(* Schneider Machine Expert - Basic project memory words, file version 2.0.0.0 *)
(* ProjectInformations: Name=New project *)

HARDWARE
  Cpu 0: TM221CE16R
  EthernetConfiguration: NetworkName=M221, IpAllocationMode=FixedAddress, IpAddress=0.0.0.0, SubnetMask=0.0.0.0
  SerialLineConfiguration: Baud=Baud19200, Parity=ParityEven, DataBits=DataBits8, StopBits=StopBits1, PhysicalMedium=PhysicalMediumRs485, TransmissionMode=TransmissionModeModbusRtu, SlaveId=1, Addressing=SlaveAddressing
  MastTask: UsePeriodScanMode=false, PeriodScan=100
  FastTask: Period=255
  CpuBehavior: StartingMode=StartAsPreviousState, AutoSaveRamOnEeprom=true, WatchdogPeriod=250

SYMBOLS  (address, symbol, comment, settings)

POU New POU
  (* SectionNumber=1 *)

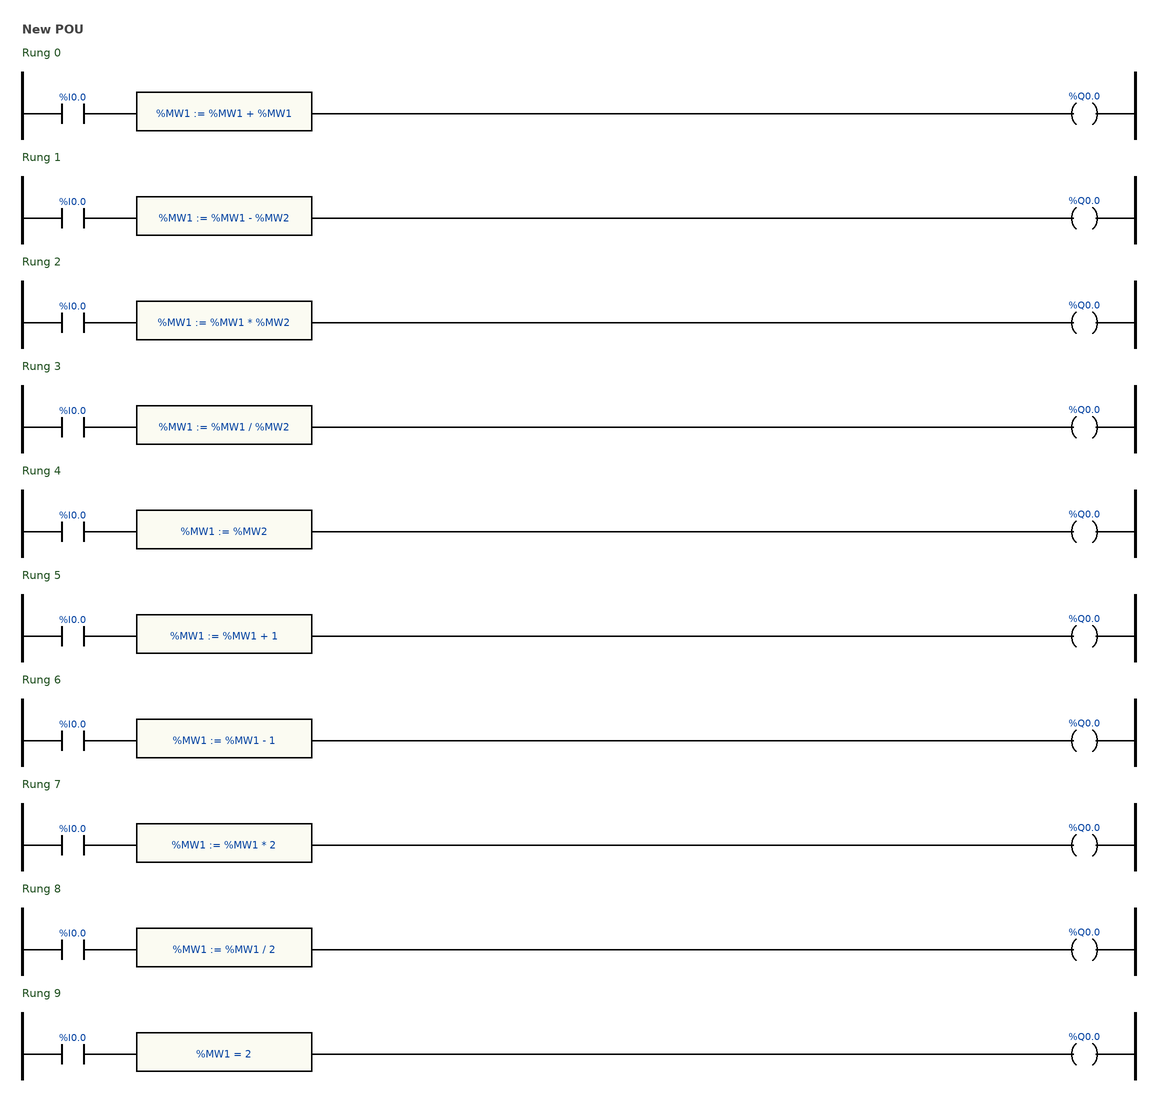

// Rung 0
  LD %I0.0
  OPER [ %MW1 := %MW1 + %MW1 ]
  ST %Q0.0
  // as ST:
  //   IF %I0.0 THEN %MW1 := %MW1 + %MW1; END_IF;
  //   %Q0.0 := %I0.0;

// Rung 1
  LD %I0.0
  OPER [ %MW1 := %MW1 - %MW2 ]
  ST %Q0.0
  // as ST:
  //   IF %I0.0 THEN %MW1 := %MW1 - %MW2; END_IF;
  //   %Q0.0 := %I0.0;

// Rung 2
  LD %I0.0
  OPER [ %MW1 := %MW1 * %MW2 ]
  ST %Q0.0
  // as ST:
  //   IF %I0.0 THEN %MW1 := %MW1 * %MW2; END_IF;
  //   %Q0.0 := %I0.0;

// Rung 3
  LD %I0.0
  OPER [ %MW1 := %MW1 / %MW2 ]
  ST %Q0.0
  // as ST:
  //   IF %I0.0 THEN %MW1 := %MW1 / %MW2; END_IF;
  //   %Q0.0 := %I0.0;

// Rung 4
  LD %I0.0
  OPER [ %MW1 := %MW2 ]
  ST %Q0.0
  // as ST:
  //   IF %I0.0 THEN %MW1 := %MW2; END_IF;
  //   %Q0.0 := %I0.0;

// Rung 5
  LD %I0.0
  OPER [ %MW1 := %MW1 + 1 ]
  ST %Q0.0
  // as ST:
  //   IF %I0.0 THEN %MW1 := %MW1 + 1; END_IF;
  //   %Q0.0 := %I0.0;

// Rung 6
  LD %I0.0
  OPER [ %MW1 := %MW1 - 1 ]
  ST %Q0.0
  // as ST:
  //   IF %I0.0 THEN %MW1 := %MW1 - 1; END_IF;
  //   %Q0.0 := %I0.0;

// Rung 7
  LD %I0.0
  OPER [ %MW1 := %MW1 * 2 ]
  ST %Q0.0
  // as ST:
  //   IF %I0.0 THEN %MW1 := %MW1 * 2; END_IF;
  //   %Q0.0 := %I0.0;

// Rung 8
  LD %I0.0
  OPER [ %MW1 := %MW1 / 2 ]
  ST %Q0.0
  // as ST:
  //   IF %I0.0 THEN %MW1 := %MW1 / 2; END_IF;
  //   %Q0.0 := %I0.0;

// Rung 9
  LD %I0.0
  AND [ %MW1 = 2 ]
  ST %Q0.0
  // as ST:
  //   %Q0.0 := %I0.0 AND %MW1 = 2;

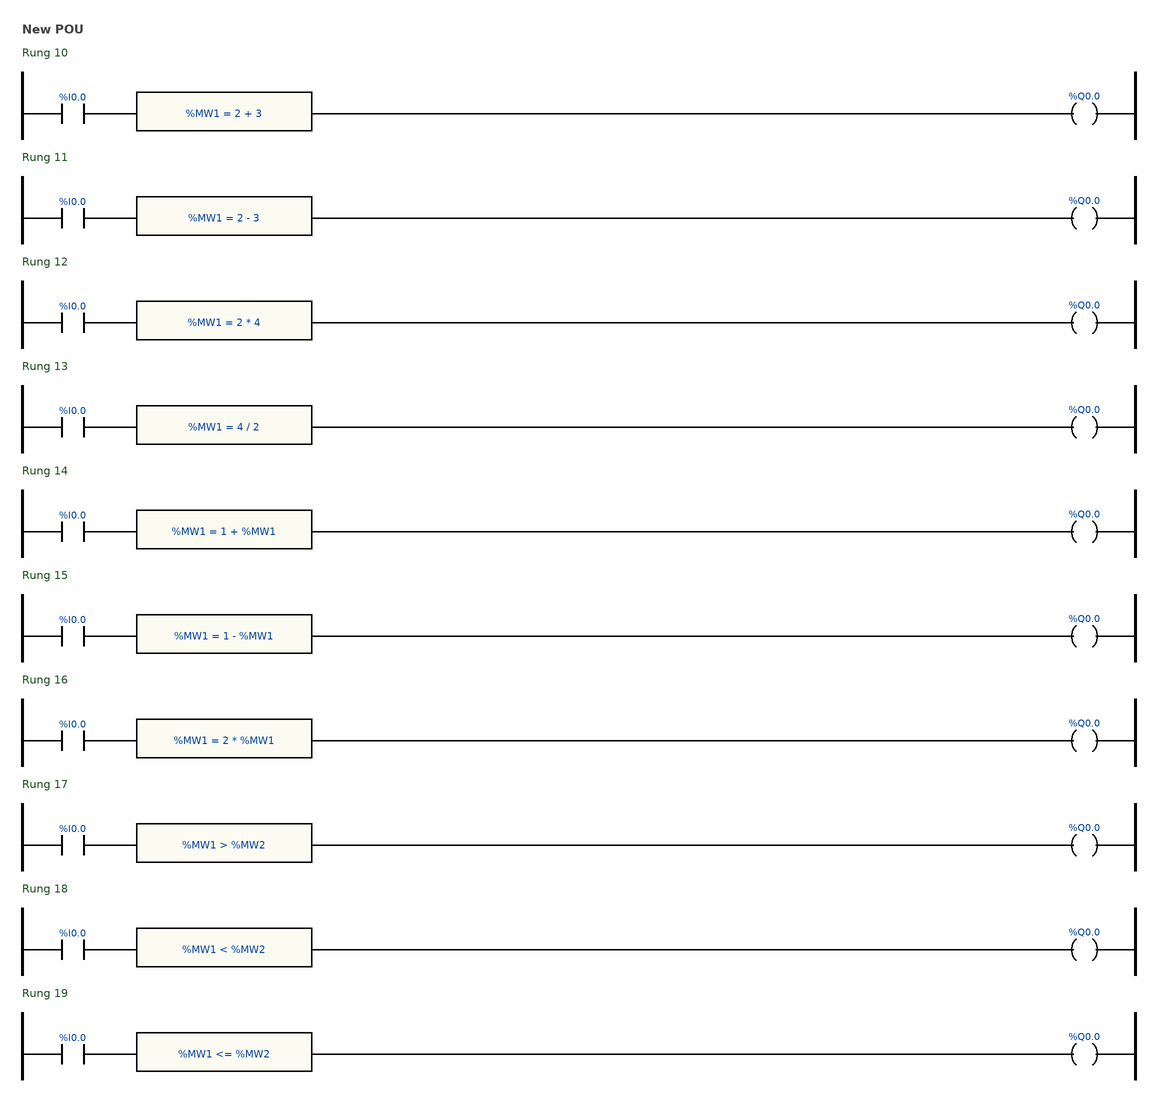

// Rung 10
  LD %I0.0
  AND [ %MW1 = 2 + 3 ]
  ST %Q0.0
  // as ST:
  //   %Q0.0 := %I0.0 AND %MW1 = 2 + 3;

// Rung 11
  LD %I0.0
  AND [ %MW1 = 2 - 3 ]
  ST %Q0.0
  // as ST:
  //   %Q0.0 := %I0.0 AND %MW1 = 2 - 3;

// Rung 12
  LD %I0.0
  AND [ %MW1 = 2 * 4 ]
  ST %Q0.0
  // as ST:
  //   %Q0.0 := %I0.0 AND %MW1 = 2 * 4;

// Rung 13
  LD %I0.0
  AND [ %MW1 = 4 / 2 ]
  ST %Q0.0
  // as ST:
  //   %Q0.0 := %I0.0 AND %MW1 = 4 / 2;

// Rung 14
  LD %I0.0
  AND [ %MW1 = 1 + %MW1 ]
  ST %Q0.0
  // as ST:
  //   %Q0.0 := %I0.0 AND %MW1 = 1 + %MW1;

// Rung 15
  LD %I0.0
  AND [ %MW1 = 1 - %MW1 ]
  ST %Q0.0
  // as ST:
  //   %Q0.0 := %I0.0 AND %MW1 = 1 - %MW1;

// Rung 16
  LD %I0.0
  AND [ %MW1 = 2 * %MW1 ]
  ST %Q0.0
  // as ST:
  //   %Q0.0 := %I0.0 AND %MW1 = 2 * %MW1;

// Rung 17
  LD %I0.0
  AND [ %MW1 > %MW2 ]
  ST %Q0.0
  // as ST:
  //   %Q0.0 := %I0.0 AND %MW1 > %MW2;

// Rung 18
  LD %I0.0
  AND [ %MW1 < %MW2 ]
  ST %Q0.0
  // as ST:
  //   %Q0.0 := %I0.0 AND %MW1 < %MW2;

// Rung 19
  LD %I0.0
  AND [ %MW1 <= %MW2 ]
  ST %Q0.0
  // as ST:
  //   %Q0.0 := %I0.0 AND %MW1 <= %MW2;

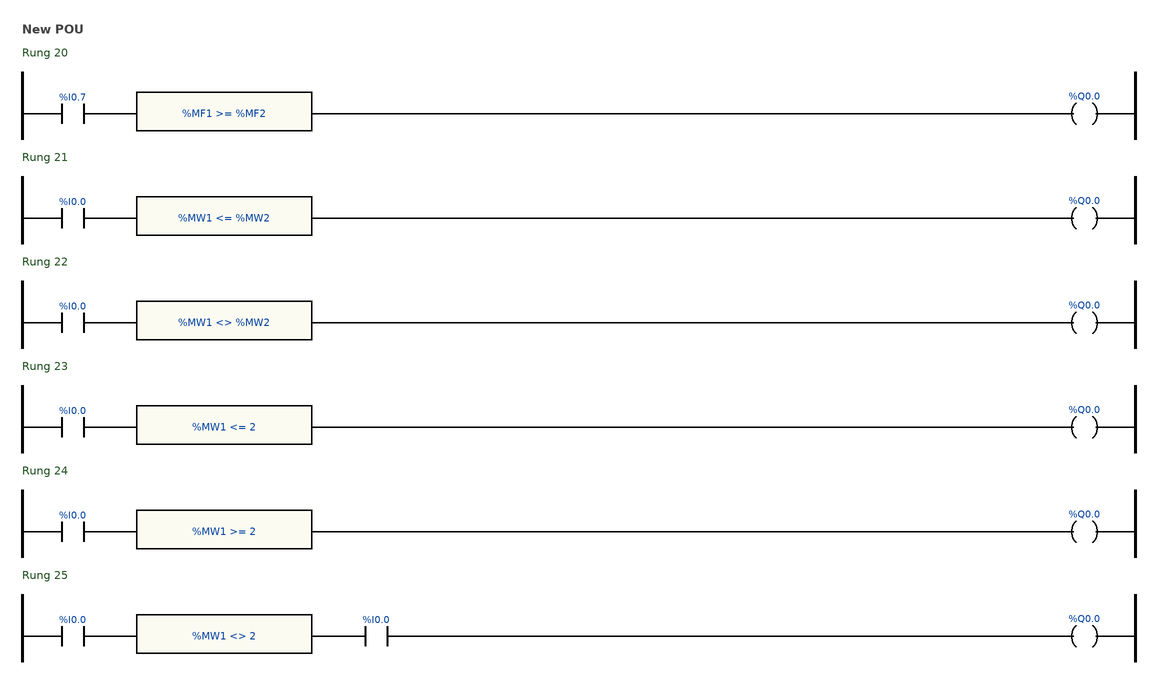

// Rung 20
  LD %I0.7
  AND [ %MF1 >= %MF2 ]
  ST %Q0.0
  // as ST:
  //   %Q0.0 := %I0.7 AND %MF1 >= %MF2;

// Rung 21
  LD %I0.0
  AND [ %MW1 <= %MW2 ]
  ST %Q0.0
  // as ST:
  //   %Q0.0 := %I0.0 AND %MW1 <= %MW2;

// Rung 22
  LD %I0.0
  AND [ %MW1 <> %MW2 ]
  ST %Q0.0
  // as ST:
  //   %Q0.0 := %I0.0 AND %MW1 <> %MW2;

// Rung 23
  LD %I0.0
  AND [ %MW1 <= 2 ]
  ST %Q0.0
  // as ST:
  //   %Q0.0 := %I0.0 AND %MW1 <= 2;

// Rung 24
  LD %I0.0
  AND [ %MW1 >= 2 ]
  ST %Q0.0
  // as ST:
  //   %Q0.0 := %I0.0 AND %MW1 >= 2;

// Rung 25
  LD %I0.0
  AND [ %MW1 <> 2 ]
  AND %I0.0
  ST %Q0.0
  // as ST:
  //   %Q0.0 := %I0.0 AND %MW1 <> 2 AND %I0.0;
